PROGRAM MAIN
VAR
END_VAR

//prg_PWM();
//prg_Click_Log();
//prg_GetMinimum();
//prg_Personeelsdata();
//prg_SearchString();
prg_Druktoets_Functies();

END_PROGRAM

(* stored: Version 1.1.0.1, ProductVersion 3.1.4024.15
   POU MAIN: Id {0936af44-c389-4e13-9d21-3adac139443b}, SpecialFunc None *)
